PROGRAM CLICK_ROUTINE

VAR_INPUT
	pushButton	:BOOL;
END_VAR

VAR_OUTPUT
	pulseOutput	:BOOL;
END_VAR

VAR
	pulse		:TP;
END_VAR

pulse(IN:= pushButton, PT:= t#500ms, Q=> pulseOutput, ET=> );

END_PROGRAM

(* stored: Version 1.1.0.1, ProductVersion 3.1.4024.13
   POU CLICK_ROUTINE: Id {0420af6a-a9b6-4312-9a7a-c27a7638216b}, SpecialFunc None *)
